(* Logix 5000 project; controller Amvex_Thorpe_Flowmeter vendor 1 type 14 code 106 rev 33.13; software revision 33.01; part 5 of 16 *)

ADD_ON_INSTRUCTION MovePose   (* revision 0.1, vendor Mecademic Inc., ExecuteEnableInFalse *)
// Move to a position relative to WRF (x-y-z in mm, a-b-c in degrees), All joints start and end movement at the same time
VAR_IN_OUT
   RobotInputs : _061D:Meca500_86BDA20B:I:0; {required}
   RobotOutputs : _061D:Meca500_01F88326:O:0; {required}
END_VAR
VAR_INPUT
   Pose_X_Pos : REAL; {required}
   Pose_Y_Pos : REAL; {required}
   Pose_Z_Pos : REAL; {required}
   Pose_rX_Ang : REAL; {required}
   Pose_rY_Ang : REAL; {required}
   Pose_rZ_Ang : REAL; {required}
   ExternalStateControl : BOOL; {required}
   ExternalMoveID : INT; {required}
END_VAR
VAR_OUTPUT
   Enabled : BOOL; {visible}
   Sent : BOOL; {visible}
   Buffered : BOOL; {visible}
   Error : BOOL; {visible}
END_VAR
VAR
   InternalMoveID : INT; {access None}
   MoveIDTrig : BOOL; {access None}
   MoveIDUpdated : BOOL; {access None}
   OneShot : DINT; {access None}
   FirstScan : BOOL; {access None}
END_VAR

ROUTINE EnableInFalse   (* ladder *)
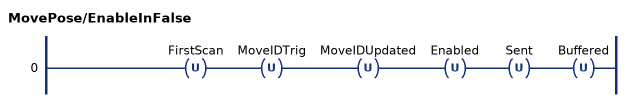
   0: OTU(FirstScan)OTU(MoveIDTrig)OTU(MoveIDUpdated)OTU(Enabled)OTU(Sent)OTU(Buffered);
END_ROUTINE

ROUTINE Logic   (* ladder *)
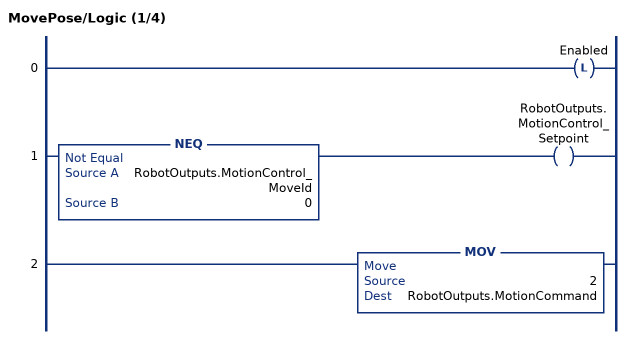
   0: OTL(Enabled);
   1: NEQ(RobotOutputs.MotionControl_MoveId,0)OTE(RobotOutputs.MotionControl_Setpoint);
   2: MOV(2,RobotOutputs.MotionCommand);
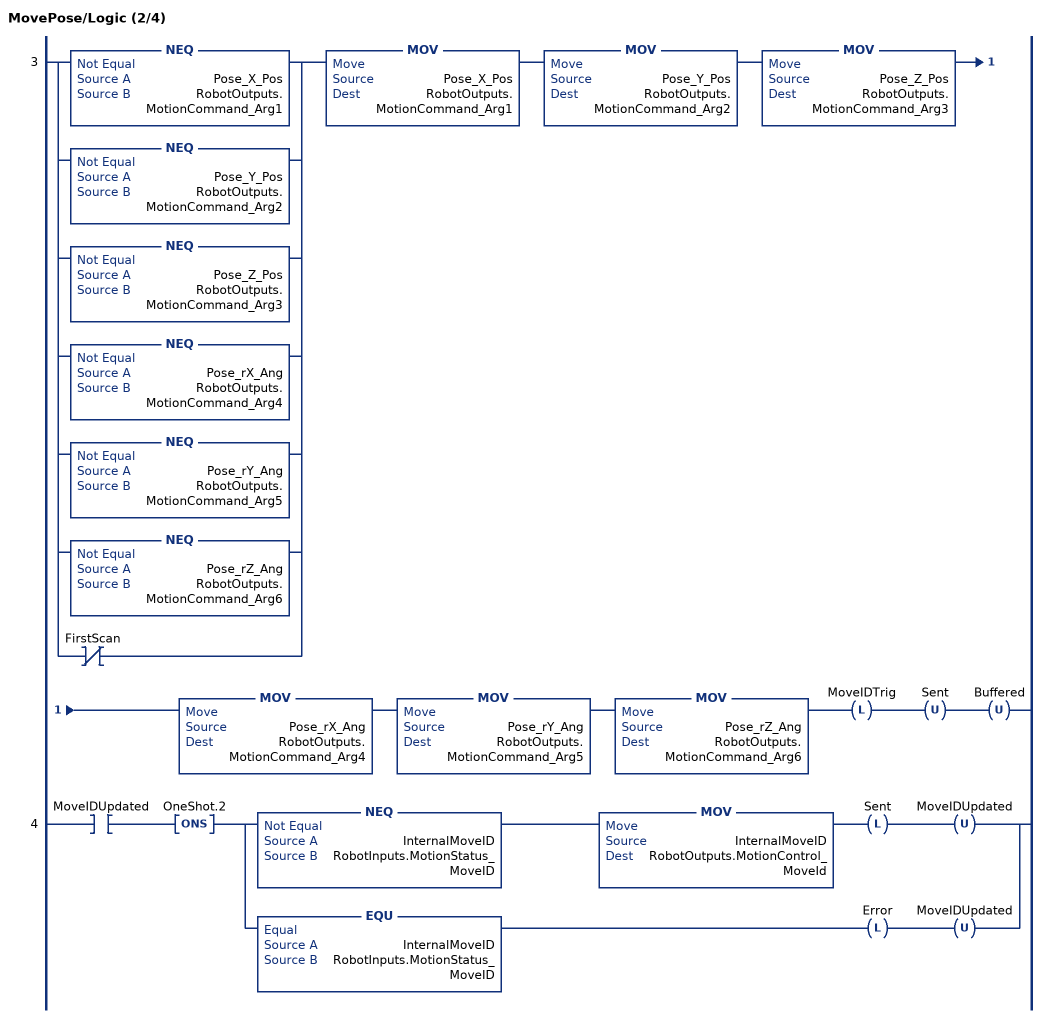
   3: [NEQ(Pose_X_Pos,RobotOutputs.MotionCommand_Arg1) ,NEQ(Pose_Y_Pos,RobotOutputs.MotionCommand_Arg2) ,NEQ(Pose_Z_Pos,RobotOutputs.MotionCommand_Arg3) ,NEQ(Pose_rX_Ang,RobotOutputs.MotionCommand_Arg4) ,NEQ(Pose_rY_Ang,RobotOutputs.MotionCommand_Arg5) ,NEQ(Pose_rZ_Ang,RobotOutputs.MotionCommand_Arg6) ,XIO(FirstScan) ]MOV(Pose_X_Pos,RobotOutputs.MotionCommand_Arg1)MOV(Pose_Y_Pos,RobotOutputs.MotionCommand_Arg2)MOV(Pose_Z_Pos,RobotOutputs.MotionCommand_Arg3)MOV(Pose_rX_Ang,RobotOutputs.MotionCommand_Arg4)MOV(Pose_rY_Ang,RobotOutputs.MotionCommand_Arg5)MOV(Pose_rZ_Ang,RobotOutputs.MotionCommand_Arg6)OTL(MoveIDTrig)OTU(Sent)OTU(Buffered);
   4: XIC(MoveIDUpdated)ONS(OneShot.2)[NEQ(InternalMoveID,RobotInputs.MotionStatus_MoveID) MOV(InternalMoveID,RobotOutputs.MotionControl_MoveId) OTL(Sent) OTU(MoveIDUpdated) ,EQU(InternalMoveID,RobotInputs.MotionStatus_MoveID) OTL(Error) OTU(MoveIDUpdated) ];
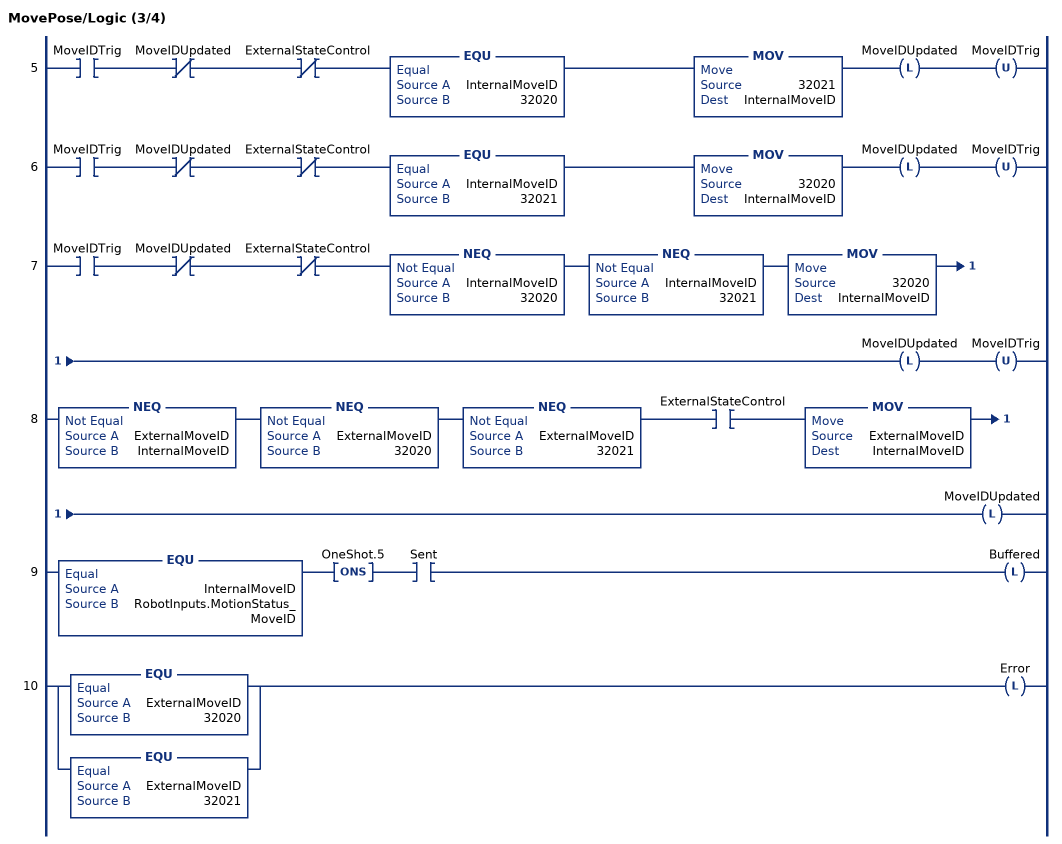
   5: XIC(MoveIDTrig)XIO(MoveIDUpdated)XIO(ExternalStateControl)EQU(InternalMoveID,32020)MOV(32021,InternalMoveID)OTL(MoveIDUpdated)OTU(MoveIDTrig);
   6: XIC(MoveIDTrig)XIO(MoveIDUpdated)XIO(ExternalStateControl)EQU(InternalMoveID,32021)MOV(32020,InternalMoveID)OTL(MoveIDUpdated)OTU(MoveIDTrig);
   7: XIC(MoveIDTrig)XIO(MoveIDUpdated)XIO(ExternalStateControl)NEQ(InternalMoveID,32020)NEQ(InternalMoveID,32021)MOV(32020,InternalMoveID)OTL(MoveIDUpdated)OTU(MoveIDTrig);
   8: NEQ(ExternalMoveID,InternalMoveID)NEQ(ExternalMoveID,32020)NEQ(ExternalMoveID,32021)XIC(ExternalStateControl)MOV(ExternalMoveID,InternalMoveID)OTL(MoveIDUpdated);
   9: EQU(InternalMoveID,RobotInputs.MotionStatus_MoveID)ONS(OneShot.5)XIC(Sent)OTL(Buffered);
   10: [EQU(ExternalMoveID,32020) ,EQU(ExternalMoveID,32021) ]OTL(Error);
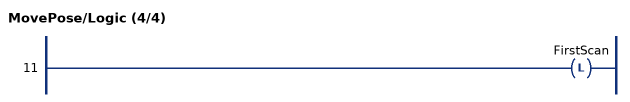
   11: OTL(FirstScan);
END_ROUTINE
END_ADD_ON_INSTRUCTION

ADD_ON_INSTRUCTION ODE3_STD   (* revision 2.1, vendor Invertek Drives Ltd. *)
// Standard ODE-3 AOI
// Revision note:
// This is an basic Add-On Instruction for controlling the Optidrive E3 drives using an OPT-2-ETHEG-IN Ethernet/IP gateway.
// Help:
// This AOI support communication with a drive at address 1 (P-36 Index 1 = 1) using the standard Data Telefram ( 4 Words In/ 4 Words Out).
// This AOI instruction can be used:
// 1. with compatible EDS file: OPC-2-ETHIG-IN_V2.63 Allen Bradley Compatible Connection.eds
// 2. in Generic Mode as an Ethernet-Bridge (Generic EtherNet/IP CIP Bridge)
// Module configuration settings:
// 1. for use with EDS
//    Connection method:  STD
//    Data type:          SINT
//    Input:                 8 SINT
//    Output:              8 SINT
// 2. Generic Mode
// Please add Ethernet-Bridge to the project and set IP Address assigned to the module/drive. Under CIP Bus please add New module/ CIP-Module.
// Settings:
// Comm Format: Data – SINT
// Address: 1 (must be the same as the drive address set in P-36 Index 1)
// Assembly Instance:
// Input:	  6	Size: 8 (8-bit)
// Output:      1	Size: 8 (8-bit)
// Config:	  2	Size: 0 (8-bit)
// RPI:            >= 50ms
// Note: In generic mode there is no support for TCP/IP connection status. Please assign temp tag (BOOL) as a DriveComStatus.
VAR_INPUT
   DriveComStatus : BOOL; {required}   // Drive Communication Status
END_VAR
VAR_IN_OUT
   DriveIn : SINT[8]; {required}   // Drive Input Tag
   DriveOut : SINT[8]; {required}   // Drive Output Tag
        [4]   // Fieldbus Ramp Time MSB
        [5]   // Fieldbus Ramp Time LSB
        [1]   // Reserved
        [0].0   // Run
        [0].1   // Fast Stop
        [2]   // Speed Reference MSB
        [3]   // Speed Reference LSB
        [0].2   // Reset
        [0].3   // Coast
        [0]   // Control Word
END_VAR
VAR_INPUT
   Run : BOOL; {required}   // Start
   Reverse : BOOL; {required}   // Run revers
   Reset : BOOL; {required}   // Trip reset (momnetary 1 to reset)
   Fast_Stop : BOOL; {required}   // Fast Stop (P-24 Ramp time)
   Coast : BOOL; {required}   // Coast to stop
END_VAR
VAR_IN_OUT
   Speed_SP : REAL; {required}   // Max 500.0Hz
   Ramp_Time : REAL; {required}   // Max 600.00s
END_VAR
VAR_OUTPUT
   Communication_Fault : BOOL; {access Read Only, visible}
   Ready : BOOL; {access Read Only, visible}   // Drive Ready (Enabled & Not Tripped)
   Running : BOOL; {access Read Only, visible}   // Drive running
   Trip : BOOL; {access Read Only, visible}   // Drive tripped
   Standby : BOOL; {access Read Only, visible}   // Drive in Standby Mode
   Fault_code : SINT; {access Read Only, visible}   // Active Fault code
   Motor_Speed : REAL; {access Read Only, visible}   // Actual speed of the motor
   Motor_Current : REAL; {access Read Only, visible}   // Ouput current
   Output_Torque : REAL; {access Read Only, visible}   // Motor torque in %
END_VAR
VAR
   int_cur : INT; {access None}
   int_spd : INT; {access None}
   int_ramp : REAL; {access None}
   int_ramp_INT : INT; {access None}
   int_spd_SP_INT : INT; {access None}
   int_spd_SP_REAL : REAL; {access None}
   int_SPD_T : INT; {access None}
   int_tq : INT; {access None}
END_VAR

ROUTINE Logic   (* ladder *)
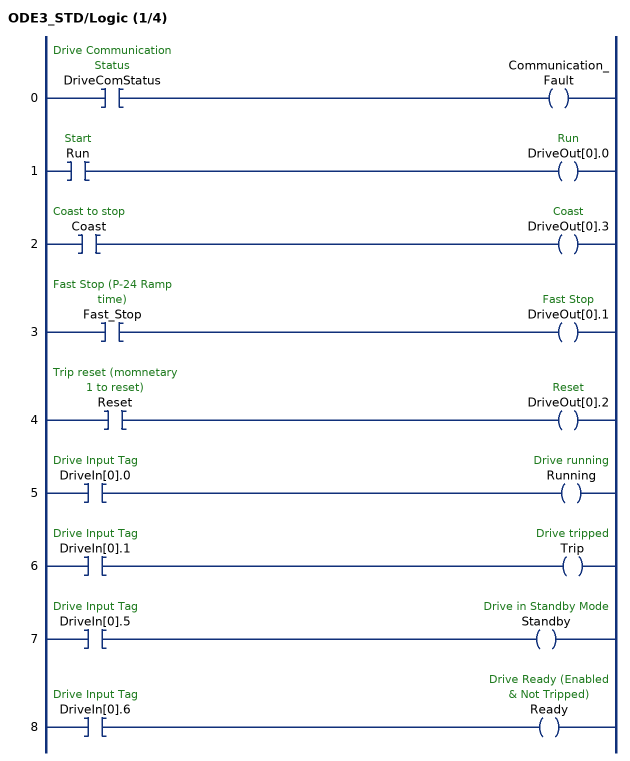
   0: XIC(DriveComStatus)OTE(Communication_Fault);
   1: XIC(Run)OTE(DriveOut[0].0);
   2: XIC(Coast)OTE(DriveOut[0].3);
   3: XIC(Fast_Stop)OTE(DriveOut[0].1);
   4: XIC(Reset)OTE(DriveOut[0].2);
   5: XIC(DriveIn[0].0)OTE(Running);
   6: XIC(DriveIn[0].1)OTE(Trip);
   7: XIC(DriveIn[0].5)OTE(Standby);
   8: XIC(DriveIn[0].6)OTE(Ready);
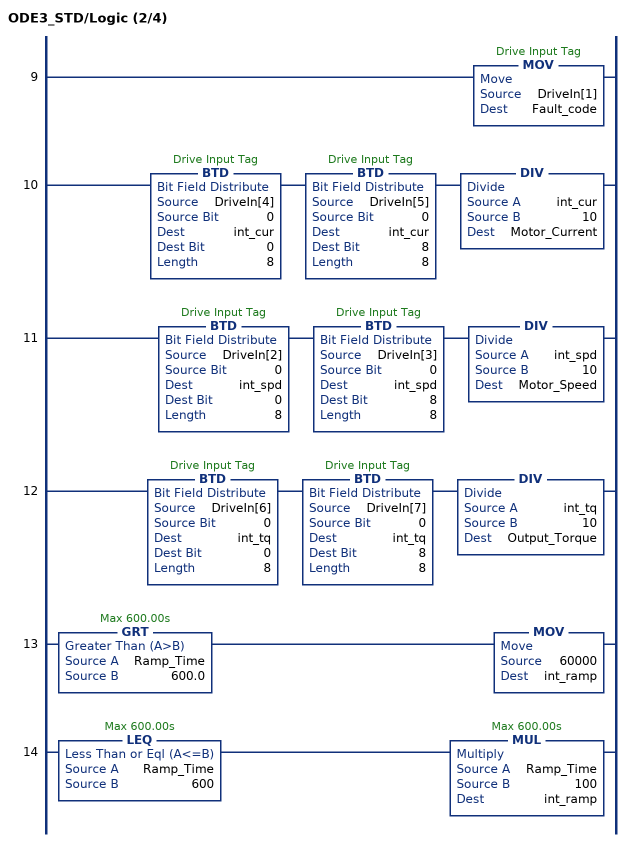
   9: MOV(DriveIn[1],Fault_code);
   10: BTD(DriveIn[4],0,int_cur,0,8)BTD(DriveIn[5],0,int_cur,8,8)DIV(int_cur,10,Motor_Current);
   11: BTD(DriveIn[2],0,int_spd,0,8)BTD(DriveIn[3],0,int_spd,8,8)DIV(int_spd,10,Motor_Speed);
   12: BTD(DriveIn[6],0,int_tq,0,8)BTD(DriveIn[7],0,int_tq,8,8)DIV(int_tq,10,Output_Torque);
   13: GRT(Ramp_Time,600.0)MOV(60000,int_ramp);
   14: LEQ(Ramp_Time,600)MUL(Ramp_Time,100,int_ramp);
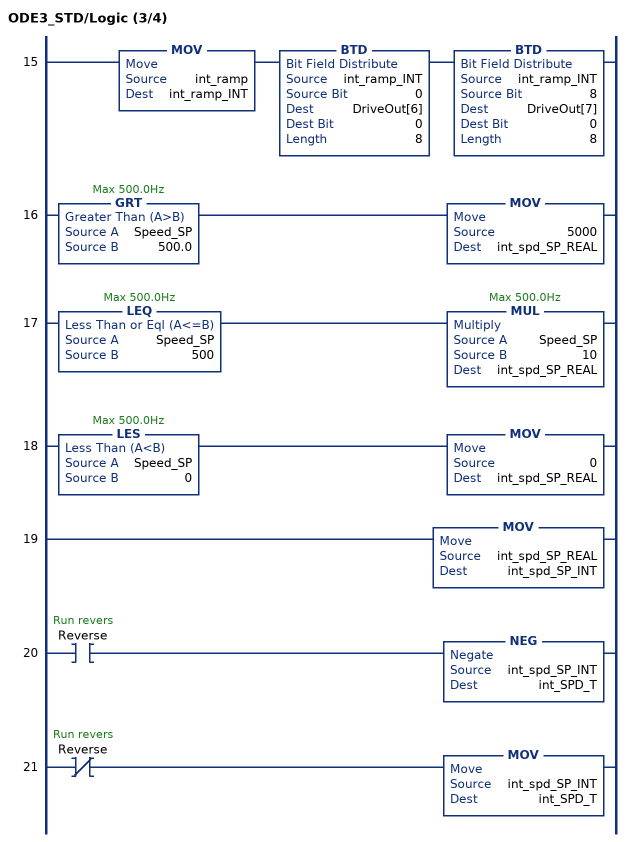
   15: MOV(int_ramp,int_ramp_INT)BTD(int_ramp_INT,0,DriveOut[6],0,8)BTD(int_ramp_INT,8,DriveOut[7],0,8);
   16: GRT(Speed_SP,500.0)MOV(5000,int_spd_SP_REAL);
   17: LEQ(Speed_SP,500)MUL(Speed_SP,10,int_spd_SP_REAL);
   18: LES(Speed_SP,0)MOV(0,int_spd_SP_REAL);
   19: MOV(int_spd_SP_REAL,int_spd_SP_INT);
   20: XIC(Reverse)NEG(int_spd_SP_INT,int_SPD_T);
   21: XIO(Reverse)MOV(int_spd_SP_INT,int_SPD_T);
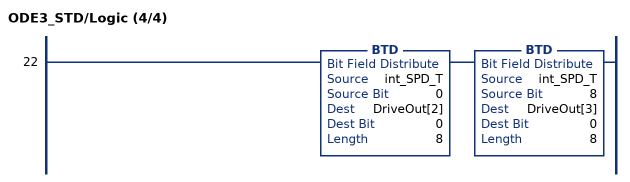
   22: BTD(int_SPD_T,0,DriveOut[2],0,8)BTD(int_SPD_T,8,DriveOut[3],0,8);
END_ROUTINE
END_ADD_ON_INSTRUCTION

ADD_ON_INSTRUCTION RobotErrors   (* revision 0.1 *)
// Meca500 errors
VAR_OUTPUT
   CommandBufferFull : BOOL; {access Read Only, visible}
   UnknownCommand : BOOL; {access Read Only, visible}
   SyntaxError : BOOL; {access Read Only, visible}
   ArgumentError : BOOL; {access Read Only, visible}
   RobotNotActivated : BOOL; {access Read Only, visible}
   RobotNotHomed : BOOL; {access Read Only, visible}
   JointOverLimit : BOOL; {access Read Only, visible}
   RobotInError : BOOL; {access Read Only, visible}
   SingularityDetected : BOOL; {access Read Only, visible}
   ActivationFailed : BOOL; {access None, visible}
   HomingFailed : BOOL; {access Read Only, visible}
   PoseOutOfReach : BOOL; {access Read Only, visible}
   CommunicationFailed : BOOL; {access Read Only, visible}
   MissingNULL : BOOL; {access Read Only, visible}
   BrakesError : BOOL; {access Read Only, visible}
   DeactivationFailed : BOOL; {access Read Only, visible}
   RobotNotSaving : BOOL; {access Read Only, visible}
   CommandNotExecutedInOfflineMode : BOOL; {access Read Only, visible}
   MasteringNeeded : BOOL; {access Read Only, visible}
   ImpossibleToReset : BOOL; {access Read Only, visible}
   DeactivationNeeded : BOOL; {access Read Only, visible}
   RobotMustBeDeactivated : BOOL; {access Read Only, visible}
   NetworkError : BOOL; {access Read Only, visible}
   MemoryFull : BOOL; {access Read Only, visible}
   AlreadySaving : BOOL; {access Read Only, visible}
   IsSaving : BOOL; {access Read Only, visible}
   GripperNotDetected : BOOL; {access Read Only, visible}
   GripperError : BOOL; {access Read Only, visible}
   AnotherUserConnected : BOOL; {access Read Only, visible}
   InitializationFailed : BOOL; {access Read Only, visible}
   HardwareProblem : BOOL; {access Read Only, visible}
   ErrorOfMotion : BOOL; {access Read Only, visible}
END_VAR
VAR_IN_OUT
   RobotInputs : _061D:Meca500_86BDA20B:I:0; {required}
   RobotOutputs : _061D:Meca500_01F88326:O:0; {required}
END_VAR
VAR_OUTPUT
   CommandTooLong : BOOL; {visible}
   ErrorSaving : BOOL; {visible}
   ErrorIsPresent : BOOL; {visible}
END_VAR

ROUTINE Logic   (* ladder *)
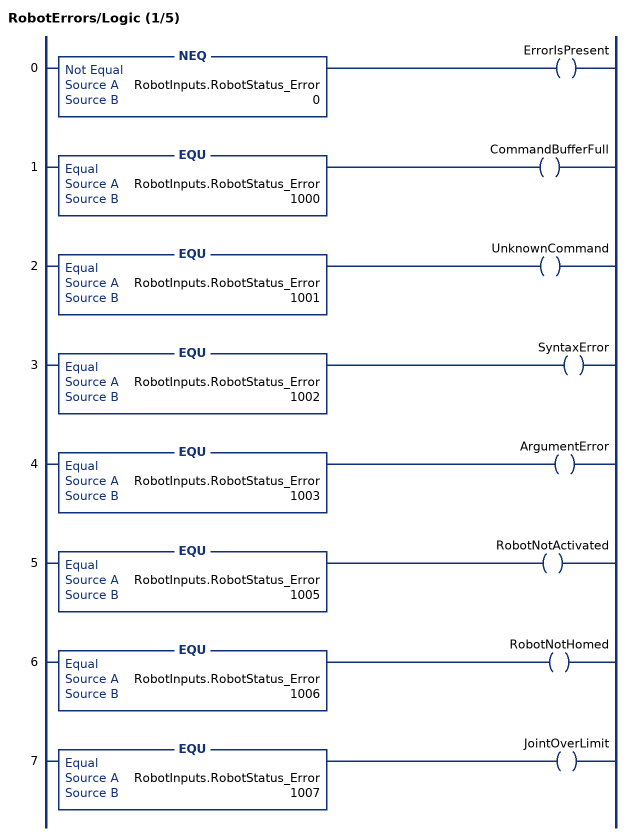
   0: NEQ(RobotInputs.RobotStatus_Error,0)OTE(ErrorIsPresent);
   1: EQU(RobotInputs.RobotStatus_Error,1000)OTE(CommandBufferFull);
   2: EQU(RobotInputs.RobotStatus_Error,1001)OTE(UnknownCommand);
   3: EQU(RobotInputs.RobotStatus_Error,1002)OTE(SyntaxError);
   4: EQU(RobotInputs.RobotStatus_Error,1003)OTE(ArgumentError);
   5: EQU(RobotInputs.RobotStatus_Error,1005)OTE(RobotNotActivated);
   6: EQU(RobotInputs.RobotStatus_Error,1006)OTE(RobotNotHomed);
   7: EQU(RobotInputs.RobotStatus_Error,1007)OTE(JointOverLimit);
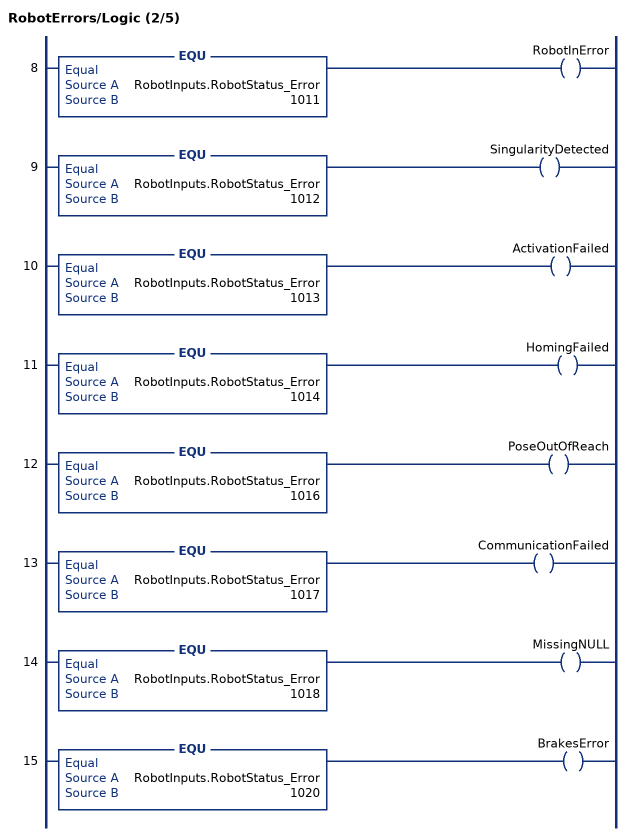
   8: EQU(RobotInputs.RobotStatus_Error,1011)OTE(RobotInError);
   9: EQU(RobotInputs.RobotStatus_Error,1012)OTE(SingularityDetected);
   10: EQU(RobotInputs.RobotStatus_Error,1013)OTE(ActivationFailed);
   11: EQU(RobotInputs.RobotStatus_Error,1014)OTE(HomingFailed);
   12: EQU(RobotInputs.RobotStatus_Error,1016)OTE(PoseOutOfReach);
   13: EQU(RobotInputs.RobotStatus_Error,1017)OTE(CommunicationFailed);
   14: EQU(RobotInputs.RobotStatus_Error,1018)OTE(MissingNULL);
   15: EQU(RobotInputs.RobotStatus_Error,1020)OTE(BrakesError);
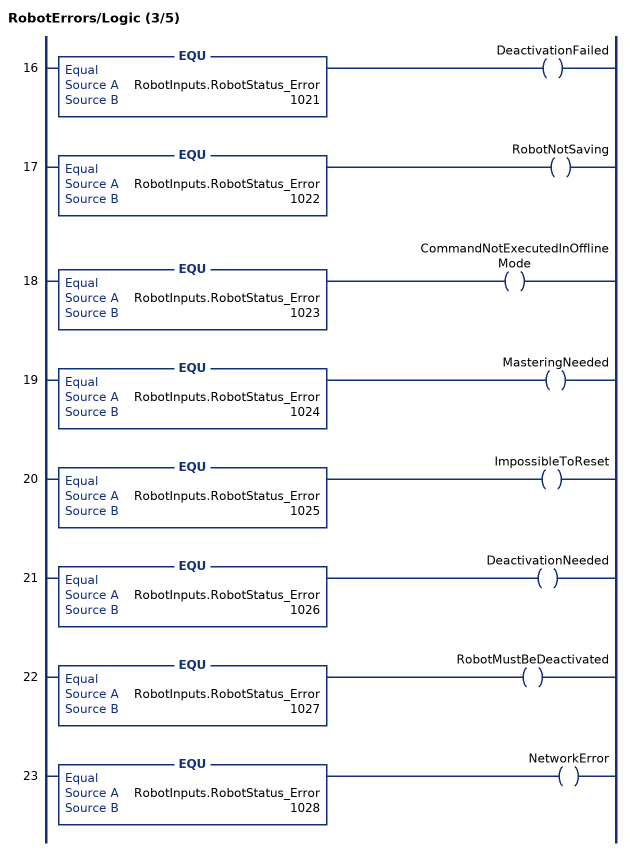
   16: EQU(RobotInputs.RobotStatus_Error,1021)OTE(DeactivationFailed);
   17: EQU(RobotInputs.RobotStatus_Error,1022)OTE(RobotNotSaving);
   18: EQU(RobotInputs.RobotStatus_Error,1023)OTE(CommandNotExecutedInOfflineMode);
   19: EQU(RobotInputs.RobotStatus_Error,1024)OTE(MasteringNeeded);
   20: EQU(RobotInputs.RobotStatus_Error,1025)OTE(ImpossibleToReset);
   21: EQU(RobotInputs.RobotStatus_Error,1026)OTE(DeactivationNeeded);
   22: EQU(RobotInputs.RobotStatus_Error,1027)OTE(RobotMustBeDeactivated);
   23: EQU(RobotInputs.RobotStatus_Error,1028)OTE(NetworkError);
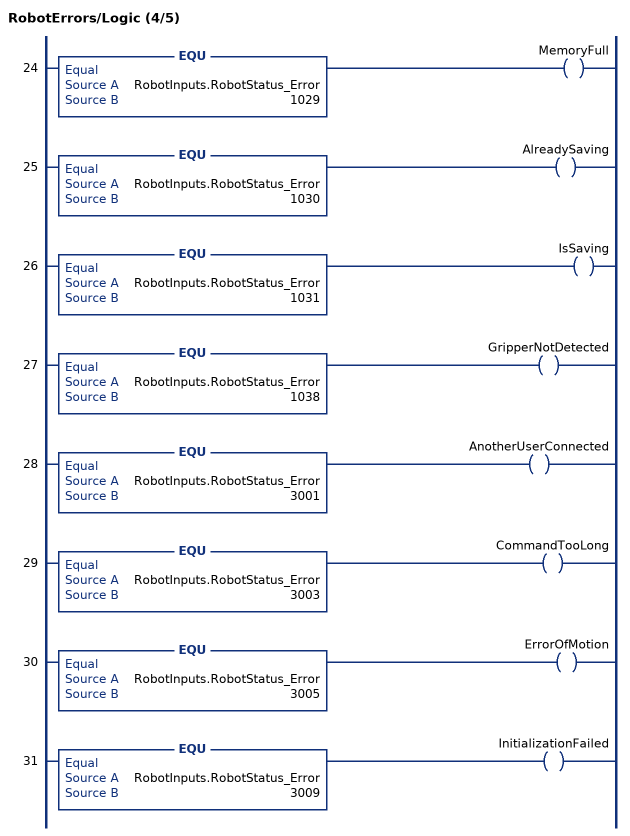
   24: EQU(RobotInputs.RobotStatus_Error,1029)OTE(MemoryFull);
   25: EQU(RobotInputs.RobotStatus_Error,1030)OTE(AlreadySaving);
   26: EQU(RobotInputs.RobotStatus_Error,1031)OTE(IsSaving);
   27: EQU(RobotInputs.RobotStatus_Error,1038)OTE(GripperNotDetected);
   28: EQU(RobotInputs.RobotStatus_Error,3001)OTE(AnotherUserConnected);
   29: EQU(RobotInputs.RobotStatus_Error,3003)OTE(CommandTooLong);
   30: EQU(RobotInputs.RobotStatus_Error,3005)OTE(ErrorOfMotion);
   31: EQU(RobotInputs.RobotStatus_Error,3009)OTE(InitializationFailed);
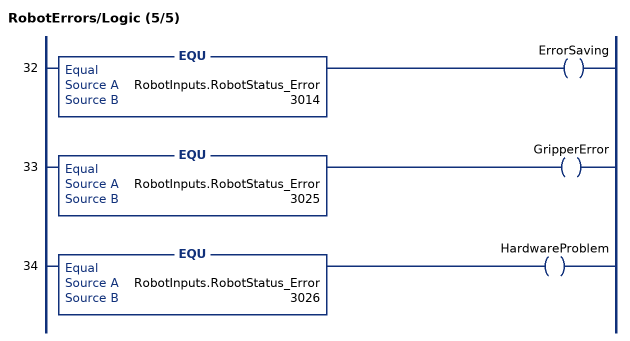
   32: EQU(RobotInputs.RobotStatus_Error,3014)OTE(ErrorSaving);
   33: EQU(RobotInputs.RobotStatus_Error,3025)OTE(GripperError);
   34: EQU(RobotInputs.RobotStatus_Error,3026)OTE(HardwareProblem);
END_ROUTINE
END_ADD_ON_INSTRUCTION

ADD_ON_INSTRUCTION SCP   (* revision 1.0 *)
VAR_INPUT
   Analog_Raw_Input : DINT; {required}
   Raw_In_Min : DINT; {required}
   Raw_In_Max : DINT; {required}
   Engineering_Min : REAL; {required}
   Engineering_Max : REAL; {required}
END_VAR
VAR_OUTPUT
   Engineered_Input_Value : REAL; {access Read Only, required}
END_VAR
VAR_INPUT
   Zero_Analog : BOOL;
END_VAR
VAR_OUTPUT
   Engineering_Offset : REAL; {access None}
END_VAR
VAR
   Scaling_Rate : REAL;
   Zero_Analog_Ons : BOOL; {access None}
   Zero_Clear_Ons : BOOL; {access None}
END_VAR

ROUTINE Logic   (* ladder *)
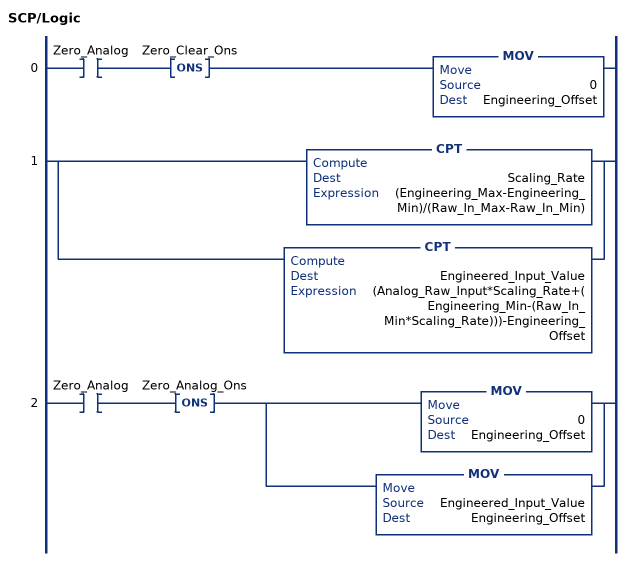
   0: XIC(Zero_Analog)ONS(Zero_Clear_Ons)MOV(0,Engineering_Offset);
   1: [CPT(Scaling_Rate,(Engineering_Max-Engineering_Min)/(Raw_In_Max-Raw_In_Min)) ,CPT(Engineered_Input_Value,(Analog_Raw_Input*Scaling_Rate+(Engineering_Min-(Raw_In_Min*Scaling_Rate)))-Engineering_Offset) ];
   2: XIC(Zero_Analog)ONS(Zero_Analog_Ons)[MOV(0,Engineering_Offset) ,MOV(Engineered_Input_Value,Engineering_Offset) ];
END_ROUTINE
END_ADD_ON_INSTRUCTION

ADD_ON_INSTRUCTION Servo_Move   (* revision 1.0, ExecuteEnableInFalse *)
VAR_IN_OUT
   Servo_Input : _0294:SV2_CM_ENETIP_63829260:I:0; {required}
        .Data[3].4   // Pos Reached
        .Data[3].2   // Zero Speed
   Servo_Output : _0294:SV2_CM_ENETIP_42190CF9:O:0; {required}
        .Data[4].0   // Trigger Path
        .Data[2].7   // Motor Stop
        .Data[3]   // Path Num
        .Data[11]   // Torque 1
        .Data[7]   // To Pos
        .Data[5]   // Speed 1
        .Data[2].2   // Torque 1
END_VAR
VAR_INPUT
   Speed : REAL; {required}
   Torque : REAL; {required}
   Position : REAL; {required}
END_VAR
VAR_OUTPUT
   Torqued : BOOL; {visible}
   DN : BOOL; {visible}
END_VAR
VAR_INPUT
   Stop : BOOL; {visible}
END_VAR
VAR_OUTPUT
   Stop_Output : BOOL; {visible}
   Trigger_Output : BOOL; {visible}
END_VAR
VAR_INPUT
   Path : INT; {required}
END_VAR
VAR
   Start_Up : BOOL; {access None}
   Torque_Treshhold : REAL; {access None}
   Trigger_TM : TIMER := (PRE := 100); {access None}
   Setup_TM : TIMER := (PRE := 50); {access None}
   Stop_TM : TIMER := (PRE := 100); {access None}
   Reset_ONS : BOOL; {access None}
   Done_TM : TIMER := (PRE := 100); {access None}
END_VAR

ROUTINE EnableInFalse   (* ladder *)
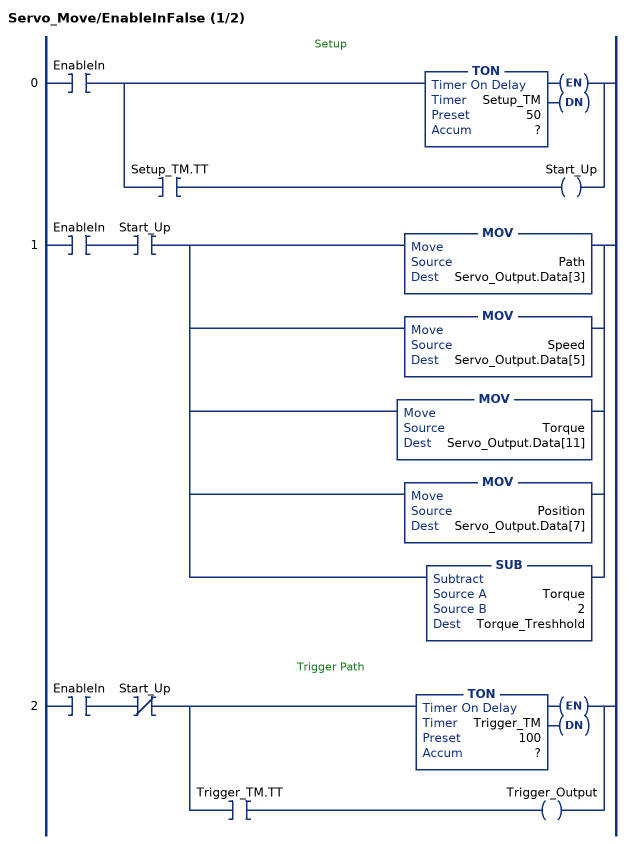
   // Setup
   0: XIC(EnableIn)[TON(Setup_TM,?,?) ,XIC(Setup_TM.TT) OTE(Start_Up) ];
   1: XIC(EnableIn)XIC(Start_Up)[MOV(Path,Servo_Output.Data[3]) ,MOV(Speed,Servo_Output.Data[5]) ,MOV(Torque,Servo_Output.Data[11]) ,MOV(Position,Servo_Output.Data[7]) ,SUB(Torque,2,Torque_Treshhold) ];
   // Trigger Path
   2: XIC(EnableIn)XIO(Start_Up)[TON(Trigger_TM,?,?) ,XIC(Trigger_TM.TT) OTE(Trigger_Output) ];
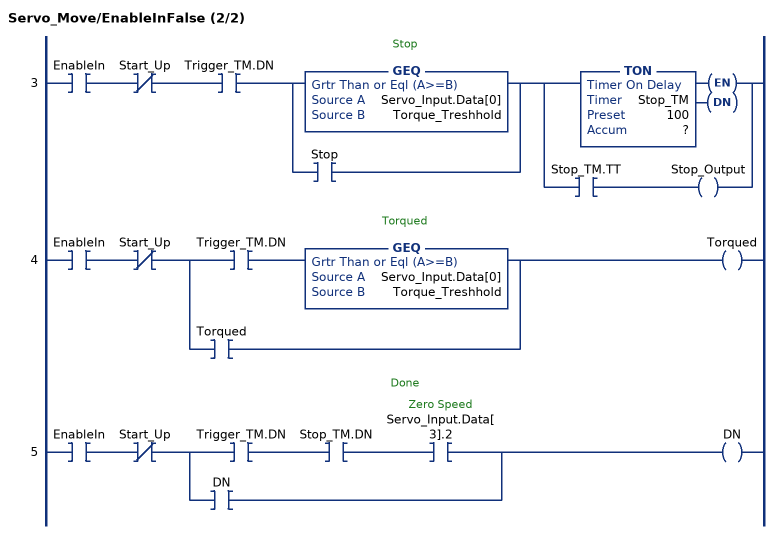
   // Stop
   3: XIC(EnableIn)XIO(Start_Up)XIC(Trigger_TM.DN)[GEQ(Servo_Input.Data[0],Torque_Treshhold) ,XIC(Stop) ][TON(Stop_TM,?,?) ,XIC(Stop_TM.TT) OTE(Stop_Output) ];
   // Torqued
   4: XIC(EnableIn)XIO(Start_Up)[XIC(Trigger_TM.DN) GEQ(Servo_Input.Data[0],Torque_Treshhold) ,XIC(Torqued) ]OTE(Torqued);
   // Done
   5: XIC(EnableIn)XIO(Start_Up)[XIC(Trigger_TM.DN) XIC(Stop_TM.DN) XIC(Servo_Input.Data[3].2) ,XIC(DN) ]OTE(DN);
END_ROUTINE

ROUTINE Logic   (* ladder *)
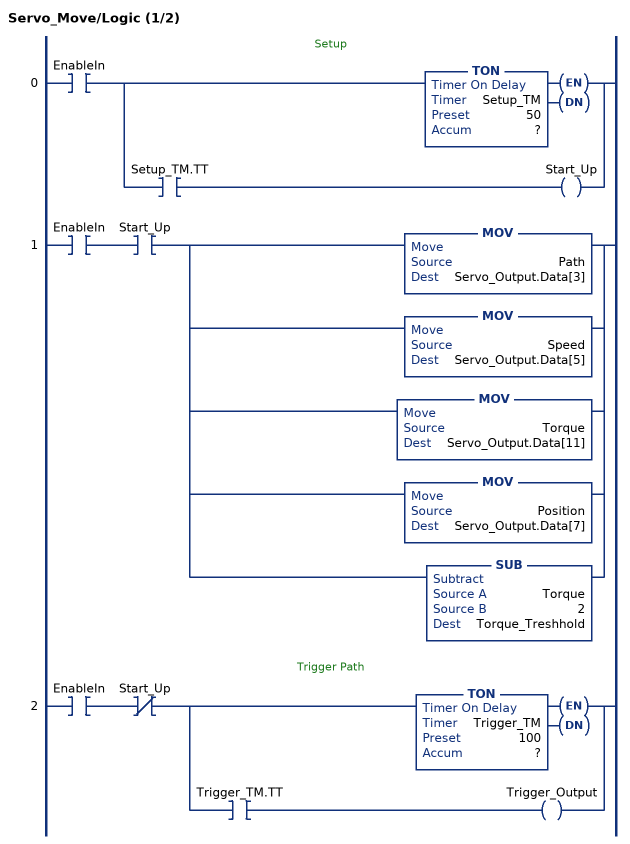
   // Setup
   0: XIC(EnableIn)[TON(Setup_TM,?,?) ,XIC(Setup_TM.TT) OTE(Start_Up) ];
   1: XIC(EnableIn)XIC(Start_Up)[MOV(Path,Servo_Output.Data[3]) ,MOV(Speed,Servo_Output.Data[5]) ,MOV(Torque,Servo_Output.Data[11]) ,MOV(Position,Servo_Output.Data[7]) ,SUB(Torque,2,Torque_Treshhold) ];
   // Trigger Path
   2: XIC(EnableIn)XIO(Start_Up)[TON(Trigger_TM,?,?) ,XIC(Trigger_TM.TT) OTE(Trigger_Output) ];
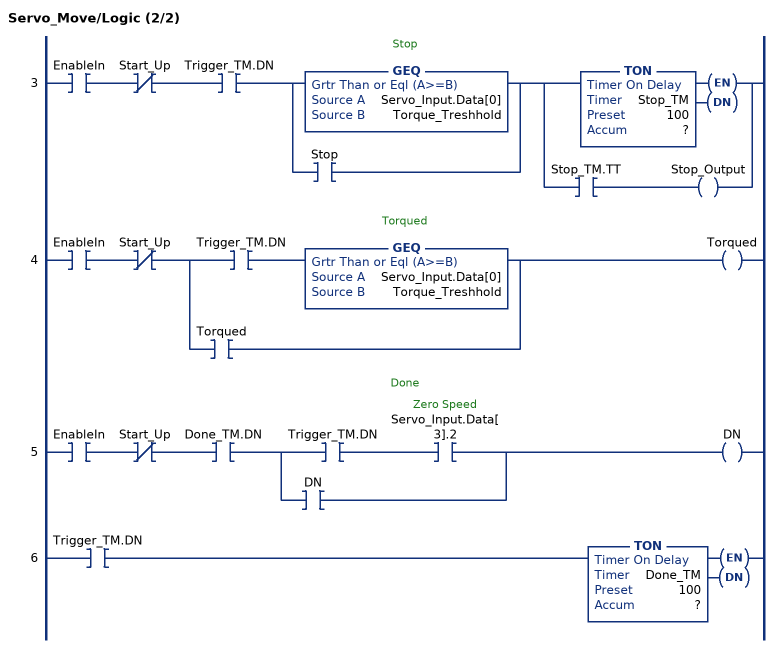
   // Stop
   3: XIC(EnableIn)XIO(Start_Up)XIC(Trigger_TM.DN)[GEQ(Servo_Input.Data[0],Torque_Treshhold) ,XIC(Stop) ][TON(Stop_TM,?,?) ,XIC(Stop_TM.TT) OTE(Stop_Output) ];
   // Torqued
   4: XIC(EnableIn)XIO(Start_Up)[XIC(Trigger_TM.DN) GEQ(Servo_Input.Data[0],Torque_Treshhold) ,XIC(Torqued) ]OTE(Torqued);
   // Done
   5: XIC(EnableIn)XIO(Start_Up)XIC(Done_TM.DN)[XIC(Trigger_TM.DN) XIC(Servo_Input.Data[3].2) ,XIC(DN) ]OTE(DN);
   6: XIC(Trigger_TM.DN)TON(Done_TM,?,?);
END_ROUTINE
END_ADD_ON_INSTRUCTION
